FUNCTION_BLOCK FB_HydThrotCir
VAR_INPUT
	//Pump
	iPump			:	I_Pump;
	//Valve
	iValve			:	I_Valve;
	//Temperatures
	iTempSup		:	I_TemperatureSensor;
	iTempRet		:	I_TemperatureSensor;
	//Controller
	iControl		:	I_HydraulicThrottlingControl;
END_VAR
VAR_OUTPUT
END_VAR
VAR
	eMode : E_ControlMode := E_ControlMode.Off;
END_VAR

PROPERTY Mode : E_ControlMode
GET
Mode := THIS^.eMode;
END_GET
SET
THIS^.eMode := Mode;
END_SET
END_PROPERTY

METHOD Run
VAR_INPUT
END_VAR
//Update temperatures
iTempSup.Run();
iTempRet.Run();

//Run components
iPump.Run();
iValve.Run();

//Run controller
iControl.Mode := eMode;
iControl.TemperatureSupAct := iTempRet.Temperature;
iControl.Run();

//Pump set properties
IF eMode = E_ControlMode.Off THEN
	iPump.SetOn := FALSE;
ELSE
	iPump.SetOn := TRUE;
END_IF
iPump.ControlMode := iControl.PumpMode;
iPump.Setpoint := iControl.PumpSet;

//Valve set properties
iValve.OpeningSetpoint := iControl.ValveSet;
END_METHOD

END_FUNCTION_BLOCK

(* stored: Version 1.1.0.1, ProductVersion 3.1.4024.3
   POU FB_HydThrotCir: Id {a08dfd34-b530-4a85-834a-60efe2b62698}, SpecialFunc None
   Property Mode: Id {8a6f300b-1743-49da-b5be-0af8720be441}
   Get Get: Id {0aaab11e-c34e-4522-8daa-fa16ac86c01e}
   Set Set: Id {79159cb7-35c9-48ec-957d-b23c5fcfd959}
   Method Run: Id {a57fc3d9-2cf3-4a7e-ab94-c5107eb69223} *)
